// TIA Portal V17 export
// export: Created 2024-09-03T21:54:54.3681033Z, ExportSetting WithDefaults, DisplayName Totally Integrated Automation Portal, DisplayVersion V17 Update 7, DisplayName TIA Portal Openness, DisplayVersion V17 Update 7, DisplayName TIA Portal Version Control Interface, DisplayVersion V17, DisplayName SINAMICS Startdrive Advanced, DisplayVersion V17 SP2, DisplayName SINAMICS Startdrive G110M, G120, G120C, G120D, G120P, G115D, DisplayVersion V17 SP2, DisplayName SINAMICS Startdrive G130, G150, S120, S150, SINAMICS MV, S210, DisplayVersion V17 SP2, DisplayName STEP 7 Professional, DisplayVersion V17 Update 7, DisplayName STEP 7 Safety, DisplayVersion V17 Update 6, DisplayName WinCC Advanced / Unified PC, DisplayVersion V17 Update 7
DATA_BLOCK "DB_MainData"   // DB5001
{ S7_Optimized_Access := 'TRUE' }
VERSION : 0.1
// stored: AutoNumber false, DBAccessibleFromOPCUA true, DBAccessibleFromWebserver true, IsOnlyStoredInLoadMemory false, IsRetainMemResEnabled false, IsWriteProtectedInAS false, MemoryReserve 100
   VAR
      SafetyLevels { S7_SetPoint := 'True'} : "UDT_SafetyLevels";
      HMI { S7_SetPoint := 'True'} : "UDT_HMI";
      ManualModeActive : Bool := FALSE;
      MachineMode : UInt := 1;   // 0= No mode active, 1= Manual mode, 2= Homing mode, 3= Automatic mode
      AntennaEdge : Bool := FALSE;
      Antenna : Bool := FALSE;
   END_VAR
BEGIN
   SafetyLevels."Level_1L+" := FALSE;
   SafetyLevels."Level_2L+" := FALSE;
   SafetyLevels."Level_3L+" := TRUE;   // Doors + safety barriers + total stop
   SafetyLevels."Level_4L+" := FALSE;   // Doors + safety barriers + total stop + light barriers
   SafetyLevels."Level_5L+" := FALSE;   // Doors + safety barriers + total stop + turn table
   SafetyLevels."Level_6L+" := FALSE;
   SafetyLevels."Level_7L+" := FALSE;
   SafetyLevels."Level_8L+" := FALSE;
   SafetyLevels."Level_9L+" := FALSE;
   SafetyLevels."Level_10L+" := FALSE;
   SafetyLevels.SystemReady := TRUE;   // Doors + safety barriers + total stop + air pressure
   HMI.ScreenData[1] := 16#0001;
   HMI.ScreenData[2] := 16#0008;
   HMI.ScreenData[3] := 16#0000;
   HMI.ScreenData[4] := 16#0007;
   HMI.ScreenData[5] := 16#0000;
   HMI.UserNumber := 0;
   HMI.ActualScreenNumber := 8;
   HMI.RequiredScreenNumber := 0;
   HMI.FunctionKeys[1..8] := FALSE;
END_DATA_BLOCK
